//enum of states
{attribute 'to_string'}
{attribute 'qualified_only'}
TYPE eTpc :
(
	//NOTE @ copy of this enum, adapt existing state names:
	TotalReset_Example,   //extra part _Example added since in the real world i've seen bugs in which scm_ programs still used eTpc in some locations. This should help prevent it.
	Initialise_Example,
	Rest_Example
)INT;
END_TYPE

//info on attributes:
//to_string			: allows the enum to be converted to string
//qualified_only 	: forces the user to start witht the type name (to avoid the situation that accidentially another enum is used)

(* stored: Version 1.1.0.1
   DUT eTpc: Id {d3d3b2c1-1eef-4965-bd65-c52c8f932a0a} *)
